{attribute addProperty BoxType "EL9222-4433-0018"}
{attribute addProperty Id "ControlAT %Q*Control_6B063D74162"}
{attribute addProperty CRC "4080052502"}
{attribute addProperty SizeInBites "16"}
{attribute addProperty SizeInBytes "2"}
TYPE OCP_Outputs_Channel_F330A916 :
STRUCT
	{attribute addProperty Name "Control"}
	Control AT %Q* : Control_6B063D74;
END_STRUCT
END_TYPE

(* stored: Version 1.2.0.0, ProductVersion 3.1.4024.9
   DUT OCP_Outputs_Channel_F330A916: Id {1f84697f-61b0-4d15-bbfd-3d405d91270a} *)
